// TIA Portal V20 export
TYPE "LER_typeAlignCalibrationConfiguration"
// stored: Access Published
   STRUCT
      MoveDistance : LReal;
   END_STRUCT;
END_TYPE
